Yaskawa INFORM job: R1_W33(0,0)KM-OK.JBI

/JOB
//NAME R1_W33(0,0)KM-OK
///FOLDERNAME KRIS-SCIANA
//POS
///NPOS 69,69,0,3,0,0
///TOOL 0
///POSTYPE PULSE
///PULSE
C00000=72256,100594,-16311,-61369,101647,63371
C00001=72256,100594,-16311,-61369,101647,63371
C00002=91745,-66930,-70045,-107044,108382,42045
C00003=88157,-70474,-71799,-106141,106049,42712
C00004=86671,-71817,-72449,-105806,105072,42972
C00005=85941,-74466,-73713,-105512,104692,43307
C00006=86671,-71817,-72449,-105806,105072,42972
C00007=84751,-71772,-72426,-105510,103718,43122
C00008=83561,-70643,-71878,-105396,102823,43103
C00009=84751,-71772,-72426,-105510,103718,43122
C00010=85686,-89844,-80471,-108137,96915,43061
C00011=85686,-89836,-80469,-108137,96914,43060
C00012=85686,-89844,-80471,-108137,96915,43061
C00013=87416,-89034,-80140,-108313,98072,42804
C00014=91641,-86743,-79187,-108837,100866,42130
C00015=90410,-65533,-69337,-70903,115869,31315
C00016=85894,-68029,-70592,-70723,112639,30963
C00017=84044,-68895,-71021,-70657,111326,30806
C00018=83406,-71048,-72074,-70470,110731,30939
C00019=84044,-68895,-71021,-70657,111326,30806
C00020=83476,-86760,-79190,-112734,99165,27043
C00021=81997,-85382,-78606,-112638,98034,27063
C00022=83476,-86760,-79190,-112734,99165,27043
C00023=85175,-86585,-79117,-112932,100310,26819
C00024=89395,-85873,-78818,-113499,103123,26219
C00025=71631,-46653,-14652,-138178,109616,-41379
C00026=71645,-31719,13616,-134693,116313,-37760
C00027=67538,-34949,9453,-135380,113683,-37157
C00028=73676,-41875,-6244,-124216,112009,-38487
C00029=66792,-34742,8732,-135645,112944,-37192
C00030=67232,-35651,8172,-135564,113244,-37248
C00031=75726,-43340,-10369,-120546,112046,-38853
C00032=75738,-39002,-1810,-119230,113443,-37473
C00033=76943,-37335,-92,-119021,114276,-37572
C00034=76943,-37335,-92,-119021,114276,-37572
C00035=75481,-38463,-509,-119021,113516,-37192
C00036=81721,-38008,-6418,-103796,114195,-36610
C00037=82250,-38825,-6921,-103667,114582,-36592
C00038=75433,-38051,224,-118919,113593,-37074
C00039=76858,-41288,-9012,-120580,112645,-39144
C00040=76858,-41288,-9012,-120580,112645,-39144
C00041=75827,-42820,-9918,-120540,112112,-38867
C00042=81717,-23054,22064,-98549,115723,-31532
C00043=82247,-23855,21516,-98352,116077,-31513
C00044=75606,-42903,-9968,-120548,111981,-38823
C00045=76873,-41376,-9063,-120574,112661,-39138
C00046=76873,-41376,-9063,-120574,112661,-39138
C00047=75623,-42896,-9961,-120548,111991,-38825
C00048=81716,-16524,33566,-96471,116069,-29580
C00049=82247,-17336,32981,-96252,116408,-29563
C00050=75773,-42789,-9656,-120480,112150,-38793
C00051=76696,-41920,-9143,-120484,112660,-39007
C00052=76696,-41920,-9143,-120484,112660,-39007
C00053=75797,-42638,-9380,-120439,112207,-38756
C00054=81717,-16601,33511,-96468,116069,-29577
C00055=82247,-17412,32926,-96249,116409,-29560
C00056=75811,-42522,-9274,-120439,112218,-38756
C00057=76900,-41013,-8379,-120470,112789,-39040
C00058=76900,-41013,-8379,-120470,112789,-39040
C00059=76185,-43664,-11862,-120837,111977,-39275
C00060=81717,-16677,33455,-96465,116070,-29574
C00061=82248,-17489,32872,-96245,116410,-29557
C00062=76141,-42332,-9146,-120428,112415,-38819
C00063=79059,-40562,-8110,-120396,114099,-39433
C00064=87960,-36038,-4572,-120572,119245,-41353
C00065=86519,-40067,-10963,-92781,74367,-28591
C00066=106744,-174057,-129458,-61191,-7105,-43025
C00067=-662,-173851,-129412,-63178,-7373,-42163
C00068=-662,-173851,-129412,-63178,-7373,-42163
BC00000=200433,1606,952938
BC00001=2104,1606,952938
BC00002=15,15,839435
BC00003=15,15,853449
BC00004=15,15,859055
BC00005=15,15,859076
BC00006=15,15,859055
BC00007=15,15,859772
BC00008=15,15,859768
BC00009=15,15,859772
BC00010=15,15,836110
BC00011=15,15,844110
BC00012=15,15,836110
BC00013=15,15,829706
BC00014=15,15,813697
BC00015=15,15,576385
BC00016=15,15,575455
BC00017=15,15,575083
BC00018=15,15,575105
BC00019=15,15,575083
BC00020=15,15,308508
BC00021=15,15,308503
BC00022=15,15,308508
BC00023=15,15,301742
BC00024=15,15,284827
BC00025=15,15,1075175
BC00026=15,15,1075175
BC00027=15,15,1075175
BC00028=15,15,1075175
BC00029=15,15,1075175
BC00030=15,15,1075175
BC00031=15,15,1075175
BC00032=15,15,1075175
BC00033=15,15,1075175
BC00034=15,15,1028712
BC00035=15,15,1028712
BC00036=15,15,1075175
BC00037=15,15,1075175
BC00038=0,15,975363
BC00039=0,707,935645
BC00040=0,707,884238
BC00041=0,707,884238
BC00042=15,15,1075175
BC00043=15,15,1075175
BC00044=0,707,828583
BC00045=0,707,828583
BC00046=0,707,776314
BC00047=0,707,776314
BC00048=15,15,1006527
BC00049=15,15,1006527
BC00050=225,707,719621
BC00051=225,707,719621
BC00052=225,707,666572
BC00053=225,707,666572
BC00054=15,15,902718
BC00055=15,15,902718
BC00056=225,707,612662
BC00057=225,707,612662
BC00058=225,707,558125
BC00059=225,707,558125
BC00060=15,15,798908
BC00061=15,15,798908
BC00062=225,707,521228
BC00063=225,707,521228
BC00064=225,707,521228
BC00065=15,15,855884
BC00066=15,207,1052077
BC00067=225820,207,1052077
BC00068=225820,484557,1052077
///POSTYPE BASE
///RECTAN
///RCONF 0,0,0,0,1,0,0,0,0,0,0,0,0,0,0,0,0,0,0,0,0,0,0,0
P00006=2.006,1.622,-0.565,0.0000,0.0000,0.0000
P00021=0.073,2.058,-0.109,0.0000,0.0000,0.0000
P00022=2.006,1.622,-0.565,0.0000,0.0000,0.0000
//INST
///DATE 2024/09/16 12:05
///ATTR SC,RW
///GROUP1 RB1,BS1
NOP
'r1_W33(0,0)
'Path S1145 (for W1147)
SFTOF
MOVJ C00000 BC00000 VJ=100.00
MOVJ C00001 BC00001 VJ=100.00
MOVJ C00002 BC00002 VJ=100.00
MOVJ C00003 BC00003 VJ=100.00
MOVL C00004 BC00004 V=60.0
REFP 3 C00005 BC00005
CALL JOB:SEARCH-R1
SET P021 P006
SFTON P021
MOVL C00006 BC00006 V=60.0
MOVL C00007 BC00007 V=60.0
REFP 3 C00008 BC00008
CALL JOB:SEARCH-R1
SET P021 P006
SFTON P021
MOVL C00009 BC00009 V=60.0
MOVL C00010 BC00010 V=60.0
REFP 3 C00011 BC00011
CALL JOB:SEARCH-R1
SET P021 P006
SFTON P021
MOVL C00012 BC00012 V=60.0
MOVL C00013 BC00013 V=166.7
MOVL C00014 BC00014 V=166.7
'Path S1146 (for W1147)
SFTOF
MOVJ C00015 BC00015 VJ=100.00
MOVJ C00016 BC00016 VJ=100.00
MOVL C00017 BC00017 V=60.0
REFP 3 C00018 BC00018
CALL JOB:SEARCH-R1
SET P022 P006
SFTON P022
MOVL C00019 BC00019 V=60.0
MOVL C00020 BC00020 V=60.0
REFP 3 C00021 BC00021
CALL JOB:SEARCH-R1
SET P022 P006
SFTON P022
MOVL C00022 BC00022 V=60.0
MOVL C00023 BC00023 V=166.7
MOVL C00024 BC00024 V=166.7
'Path W1147
SFTOF
MOVJ C00025 BC00025 VJ=100.00
SFTON P021
CALL JOB:COFNIJ_DRUT
MOVJ C00026 BC00026 VJ=100.00
MOVJ C00027 BC00027 VJ=100.00
MOVL C00028 BC00028 V=100.0 PL=0
REFP 1 C00029 BC00029
REFP 2 C00030 BC00030
MACRO1 MJ#(0) ARGF10
ARCON
MOVL C00031 BC00031 V=10.8
MOVL C00032 BC00032 V=10.8
ARCOF
MOVL C00033 BC00033 V=100.0
MOVL C00034 BC00034 V=100.0
MOVL C00035 BC00035 V=100.0 PL=0
REFP 1 C00036 BC00036
REFP 2 C00037 BC00037
MACRO1 MJ#(0) ARGF10
ARCON
MOVL C00038 BC00038 V=10.8
ARCOF
'COMMENT
MOVL C00039 BC00039 V=100.0
MOVL C00040 BC00040 V=100.0
MOVL C00041 BC00041 V=100.0 PL=0
REFP 1 C00042 BC00042
REFP 2 C00043 BC00043
MACRO1 MJ#(0) ARGF10
ARCON
'X+
MOVL C00044 BC00044 V=10.8
ARCOF
MOVL C00045 BC00045 V=100.0
SFTON P022
MOVL C00046 BC00046 V=100.0
MOVL C00047 BC00047 V=100.0 PL=0
REFP 1 C00048 BC00048
REFP 2 C00049 BC00049
MACRO1 MJ#(0) ARGF10
ARCON
MOVL C00050 BC00050 V=10.8
ARCOF
MOVL C00051 BC00051 V=100.0
MOVL C00052 BC00052 V=100.0
MOVL C00053 BC00053 V=100.0 PL=0
REFP 1 C00054 BC00054
REFP 2 C00055 BC00055
MACRO1 MJ#(0) ARGF10
ARCON
MOVL C00056 BC00056 V=10.8
ARCOF
MOVL C00057 BC00057 V=100.0
MOVL C00058 BC00058 V=100.0
MOVL C00059 BC00059 V=100.0 PL=0
REFP 1 C00060 BC00060
REFP 2 C00061 BC00061
MACRO1 MJ#(0) ARGF10
ARCON
MOVL C00062 BC00062 V=10.8
ARCOF
MOVL C00063 BC00063 V=166.7
SFTOF
MOVJ C00064 BC00064 VJ=100.00
MOVJ C00065 BC00065 VJ=100.00
MOVJ C00066 BC00066 VJ=100.00
MOVJ C00067 BC00067 VJ=100.00
MOVJ C00068 BC00068 VJ=100.00
END
